# B&R Automation Studio project rt8201
Automation Studio 4.2.9.65 SP

## Configuration Config1

CPU X20CP1381, AutomationRuntime B4.26, Build 4.1.2, Vc V4.26.1

CPU X20CP1381-RT, AutomationRuntime B4.26, Build 4.1.2, Vc V4.26.1

### Task classes (Cpu.sw)
```
Cyclic#1 (cycle 2000 us, tolerance 200000 us):
  Program1 <- Program1.prg
Binaries: TCData, arconfig, asfw, ashwd, iomap, User, Role, sysconf
ReActionTechnologyObjects: Program <- Program.prg
Libraries: AsIORTI, astime, asieccon, runtime
```

### Task classes (Cpu.sw)
```
Cyclic#1 (cycle 2000 us, tolerance 200000 us):
  sin_genera <- sin_generator.prg
  phase_loc1 <- phase_lock.prg
  rt_driver <- rt_driver.prg
VcDataObjects: Visu <- Visu.dob
Binaries: vcfile, vcrt, vcfntttf, vcctext, arial, vcmgr, vcpkat, vccovl, vccnum, vcpfar00, vcdsint, vcpfx20, vcpdvnc, vcshared, vcpdsw, vcalarm, vccbtn, vcgclass, vcdsloc, arialbd, vcnet, Visu02, TCData, vctcal, Visu01, Visu03, vccbmp, vcbclass, User, ashwd, arconfig, sysconf, Role, asfw, iomap
ReActionTechnologyObjects: phase_lock <- phase_lock.prg
Libraries: AsIORTI, fileio, asieccon, dataobj, ashw, vcresman, astime, runtime
```

### Hardware
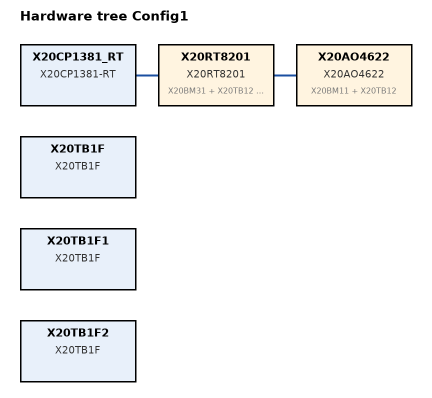
```
X20AO4622 : X20AO4622 v1.0.6.1  [SS1 -> X20TB12b.SS; SL -> X20BM11.SL1]
X20BM11 : X20BM11 v1.0.0.1  [X2X1 -> X20BM31.X2X2]
X20BM31 : X20BM31 v1.0.0.1  [X2X1 -> X20CP1381_RT.IF6]
X20CP1381_RT : X20CP1381-RT v1.3.0.0  [X1 -> X1.SL; X2 -> X2.SL; X3 -> X3.SL]
  Module X1 (Type=X1, Virtual=true, Version=1.0.0.0)
    Connection (Connector=SS1, TargetModule=X20TB1F, TargetConnector=SS)
    Connection (Connector=SL, TargetModule=X20CP1381_RT, TargetConnector=X1)
  Module X2 (Type=X2, Virtual=true, Version=1.0.0.0)
    Connection (Connector=SS1, TargetModule=X20TB1F1, TargetConnector=SS)
    Connection (Connector=SL, TargetModule=X20CP1381_RT, TargetConnector=X2)
  Module X3 (Type=X3, Virtual=true, Version=1.0.0.0)
    Connection (Connector=SS1, TargetModule=X20TB1F2, TargetConnector=SS)
    Connection (Connector=SL, TargetModule=X20CP1381_RT, TargetConnector=X3)
  Connector IF2:
    ActivateDevice = 1
    Mode = Manual
    InternetAddress = 192.168.0.10
    SubnetMask = 255.255.255.0
    Vnc1
    VncVcObjectName1 = Visu
    VncKeyMappingFile1 = VC\PS2-Keyboard.dis
  Connector IF3:
    ActivatePowerlink = 0
    CycleTime = 2000
  ConfigurationID = rt8201_Config1
  TimerDeviceType = SWIOTIMER
  SystemTick = 2000
  TaskClassIdleTime = 2000
  Cyclic1Duration = 2000
  Cyclic1Tolerance = 200000
  Cyclic2Duration = 10000
  Cyclic2Tolerance = 200000
  Cyclic3Duration = 50000
  Cyclic3Tolerance = 50000
  Cyclic4Duration = 100000
  Cyclic4Tolerance = 100000
  Cyclic5Duration = 200000
  Cyclic5Tolerance = 200000
  Cyclic6Duration = 500000
  Cyclic6Tolerance = 500000
  Cyclic7Duration = 1000000
  Cyclic7Tolerance = 1000000
  Cyclic8Duration = 10000
  Cyclic8Tolerance = 30000000
  ReActionTaskDisabled = FALSE
X20RT8201 : X20RT8201 v1.1.0.0  [SS1 -> X20TB12.SS; SS2 -> X20TB12a.SS; SL -> X20BM31.SL1]
  ReActionTask = phase_lock
  ReActionTaskDisabled = FALSE
  ReActionCycleCounter = on
  ReActionCycleTimeMin = on
  TypeRes1 = DINT
  TypeRes2 = DINT
X20TB12 : X20TB12 v1.0.0.0
X20TB12a : X20TB12 v1.0.0.0
X20TB12b : X20TB12 v1.0.0.0
X20TB1F : X20TB1F v1.0.0.0
X20TB1F1 : X20TB1F v1.0.0.0
X20TB1F2 : X20TB1F v1.0.0.0
```

### IoMap.iom - X20CP1381/IoMap.iom
```iecst
VAR_CONFIG
	::Program1:sin_val AT %QW."X20AO4622".AnalogOutput01;
	::Program1:RTCycleCounter AT %IW."X20RT8201".RTCycleCounter;
	::Program1:di1 AT %IX."X1".DigitalInput01;
END_VAR
```

### IoMap.iom - X20CP1381_RT/IoMap.iom
```iecst
VAR_CONFIG
	::rt_driver:RTCycleCounter AT %IW."X20RT8201".RTCycleCounter;
	::sin_genera:sin_val AT %QW."X20AO4622".AnalogOutput01;
	::rt_driver:RTEnable AT %QX."X20RT8201".RTEnable;
	Cyclic#1.::rt_driver:RES01 AT %ID."X20RT8201".RES01;
	::rt_driver:RES02 AT %ID."X20RT8201".RES02;
END_VAR
```

## Logical view

Binary libraries used (declarations not repeated): operator, runtime, astime, AsIecCon, AsIORTI, standard, brsystem

### Global.var - Global variables
```iecst
VAR
	sin_val_dint : DINT;
END_VAR
```


### Program Logical/phase_lock (ReAction)

#### Variables.var
```iecst
VAR
	rtiAin_0 : rtiAin;
	rtiComp_0 : rtiComp;
	rtiDout_0 : rtiDout;
	rtiDout_1 : rtiDout;
	rtiNot_0 : rtiNot;
	rtiSRff_0 : rtiSRff;
	rtiVarWrite_0 : rtiVarWrite;
	rtiVarRead_0 : rtiVarRead;
	rtiComp_1 : rtiComp;
	rtiVarWrite_1 : rtiVarWrite;
	rtiTDel_0 : rtiTDel;
	rtiRes_0 : rtiRes;
	rtiRes_1 : rtiRes;
END_VAR
```

- Cyclic.rti (not shown)

### Program Logical/sin_generator (IEC)

#### Cyclic.st - Cyclic code
```iecst
PROGRAM _INIT

	//precompute SIN table
	twoPi := 2*3.1415926;

	FOR cycle := 0 TO 9 DO
		sinTable[cycle] := REAL_TO_INT(32000 * SIN(cycle*twoPi/10));
	END_FOR

END_PROGRAM

PROGRAM _CYCLIC

	//50Hz generator
	cycle := cycle + 1;
	IF cycle > 9 THEN
		cycle := 0;
	END_IF

	sin_val := sinTable[cycle];

	sin_val_dint := sin_val;

END_PROGRAM
```

#### Variables.var - Local variables
```iecst
VAR
	twoPi : REAL;
	sinTable : ARRAY[0..19] OF INT;
	cycle : INT;
	sin_val : INT;
END_VAR
```

### Program Logical/rt_driver (IEC)

#### Cyclic.st - Cyclic code
```iecst
PROGRAM _INIT

	RTEnable := TRUE;
	pulseLength := 0.2;

	//just variable declarations
	RTCycleCounter;
	RES01;//odpovedi z RT karty do PLC
	RES02;
	RES03;
	RES04;
	RES05;
	RES06;

	time1 := 2;//cas pred svarovanim
	time2 := 1;//cas po svarovani
	period1 := 3;//kolik period se vzrustajicim vykonem
	period2 := 7;//kolik period s konstantnim vykonem
	percent1 := 40;//pocatecni vykon
	percent2 := 54;//konecny vykon

	RTInfo_0(enable := TRUE);//pro zjisteni task class

END_PROGRAM

PROGRAM _CYCLIC

	//pulse counter
	periodCounter := RES02;//citac period

	CASE step OF
		0:
			percent := 0;

			//wait for start button
			IF cmdStart THEN
				usCounter := 0;
				step := step + 1;
			END_IF
		1:
			//wait time1
			usCounter := usCounter + RTInfo_0.cycle_time;
			IF usCounter > REAL_TO_UDINT(time1 * 1000000) THEN
				period := 0;
				step := step + 1;
			END_IF

		2:
			//increase power
			IF periodCounter <> oldPeriodCounter THEN
				percent := percent1 + period * (percent2 - percent1)/period1;
				period := period + 1;
				IF period > period1 THEN
					step := step + 1;
				END_IF
			END_IF

		3:
			//hold power
			IF periodCounter <> oldPeriodCounter THEN
				period := period + 1;
				IF period > period1 + period2 THEN
					percent := 0;
					usCounter := 0;
					step := step + 1;
				END_IF
			END_IF

		4:
			//wait time2
			usCounter := usCounter + RTInfo_0.cycle_time;
			IF usCounter > REAL_TO_UDINT(time2 * 1000000) THEN
				step := 0;
			END_IF

	END_CASE

	oldPeriodCounter := periodCounter;

	//send opening angle to thyristor
	PAR01 := REAL_TO_DINT(1000000 - 10000 * percent) + 1; //1 se přičíta aby fungoval rtiDoutTime
	IF PAR01 < 1 THEN
		PAR01 := 1;
	END_IF

	//send pulse length to thyristor
	PAR02 := REAL_TO_DINT(1000000 * pulseLength);
	IF PAR02 < 0 OR PAR01 > 1000000 THEN
		PAR02 := 0;
	END_IF

END_PROGRAM
```

#### Variables.var - Local variables
```iecst
VAR
	RTCycleCounter : UINT;
END_VAR
VAR RETAIN
	time1 : REAL;
	time2 : REAL;
	period1 : INT;
	period2 : INT;
	percent1 : INT;
	percent2 : INT;
END_VAR
VAR
	RTEnable : BOOL;
	RES02 : DINT;
	RES01 : DINT;
END_VAR
```

#### Init.st - not listed in the package file held
```iecst
PROGRAM _INIT

	RTEnable := TRUE;

	//just variable declarations
	RTCycleCounter;
	RES01;

	time1;
	time2;
	period1;
	period2;
	percent1;
	percent2;

END_PROGRAM
```

- Visualisation Logical/Visu (not shown)

### Program Logical/Program (ReAction)

- Cyclic.rti - Cyclic code (not shown)

#### Variables.var - Local variables
```iecst
VAR
	rtiAin_0 : rtiAin;
	rtiRes_0 : rtiRes;
	rtiComp_0 : rtiComp;
	rtiRes_1 : rtiRes;
	rtiAnLimit_0 : rtiAnLimit;
	rtiDout_0 : rtiDout;
END_VAR
```

### Program Logical/Program1

#### Init.st
```iecst
PROGRAM _INIT
	RTCycleCounter;

END_PROGRAM
```

Listed in the project but not available here: Logical/Global.typ, Logical/sin_generator/Init.st, Logical/sin_generator/Exit.st, Logical/sin_generator/Types.typ, Logical/rt_driver/Types.typ, Logical/Program/Types.typ
